FUNCTION_BLOCK FB_AxisManager
VAR
END_VAR

END_FUNCTION_BLOCK

(* stored: Version 1.1.0.1, ProductVersion 3.1.4026.18
   POU FB_AxisManager: Id {a5239ea1-599b-4572-87dc-e1890577acbf}, SpecialFunc None *)
